FUNCTION_BLOCK FB_BeamParameterArbiter
VAR_INPUT
END_VAR
VAR_OUTPUT
	//Minimum required attenuation
	fReqAtt	:	REAL := 100; //%
END_VAR
VAR
	// List of FB asserting
	// List of assertion codes (these correlate with fault db entries)
	
	//Attenuation Request Array
	
	indexAttMax: INT;
	// Greatest attenuation requested
	fMaxReqAtt: REAL := 100;
END_VAR
VAR CONSTANT
	MAX_REQ_ARRAY	:	INT := 500;
END_VAR

(*
Beam Parameter Arbiter
A. Wallace
2018-5-18

Use the action summary blocks to hook your assertion line into the arbiter.

*)


//Attenuation
///////////////////////////////////
AttSum();

METHOD AssertBeamParameter : BOOL
VAR_INPUT
	//Parameter
	fParam	:	REAL;
	//Parameter type
	fParamType	:	E_BeamParamTyp;

END_VAR
END_METHOD

ACTION AttSum:

fMaxReqAtt	:= 100;
FOR indexAttMax := 0 TO MAX_REQ_ARRAY BY 1 DO;
	fMaxReqAtt := MAX(a
END_FOR
END_ACTION

END_FUNCTION_BLOCK

(* stored: Version 1.1.0.1, ProductVersion 3.1.4022.6
   POU FB_BeamParameterArbiter: Id {5ddfa986-ab86-4b19-bce0-591aed3e802e}, SpecialFunc None
   Method AssertBeamParameters: Id {4a784ee2-ab29-4a04-8e41-5149afa61c64}
   Action AttSum: Id {0fa0240e-bc82-4ac8-a068-21139437fa50} *)
